Universal Robots PolyScope program: mt.urp

Program mt (installation=default directory=/programs createdIn=3.8.0.61336 lastSavedIn=3.8.0.61336 robotSerialNumber=2018359174)
Calibrated DH parameters: a=[0.000103, -0.165236, -0.391809, -0.000008, 0.000072, 0]; d=[0.08937, 126.180413, -125.613724, -0.456703, 0.094787, 0.082637]; alpha=[1.569508, -0.003108, -0.027037, 1.57048, -1.570735, 0]; deltaTheta=[0, -1.172139, 1.133037, 0.038915, 0.000034, 0.000049]
Robot Program (runOnlyOnce=false)
  var_1 := p[0.0,0.0,0.0,0.0,0.0,0.0]
  Plane_1 := p[0,0,0,0,0,0]
  Base := p[0,0,0,0,0,0]
  Script file /programs/X0.script
    | address="192.168.221.2"
    | port=3000
    | sname="mt"
    | socket_open(address,port,sname)
    | p=get_actual_tcp_pose()
    | socket_send_line("X0()",sname)
    | ret=socket_read_line(sname)
    | socket_close(sname)
    | if (ret != "OK"):
    |   popup(ret,title="X0",blocking=True)
    | end
  MoveJ speed 60 deg/s, acceleration 80 deg/s^2 (useActiveTCP=true)
    Waypoint CapturePoint_1: TCP in base x=190.539 y=-105.512 z=739.544 mm, rx=-2.169 ry=2.1248 rz=-0.097 rad; joints [0.073, -70.662, -54.312, -138.221, 90.524, 0.198] deg
  Wait Sleep waitTime=1
  Script file /programs/X1.script
    | address="192.168.221.2"
    | port=3000
    | sname="mt"
    | timeout=10
    | socket_open(address,port,sname)
    | p=get_actual_tcp_pose()
    | rpy=rotvec2rpy([p[3],p[4],p[5]])
    | socket_send_string("X1(",sname)
    | socket_send_string(p[0]*1000.,sname)
    | socket_send_string(",",sname)
    | socket_send_string(p[1]*1000.,sname)
    | socket_send_string(",",sname)
    | socket_send_string(p[2]*1000.,sname)
    | socket_send_string(",",sname)
    | socket_send_string(r2d(rpy[0]),sname)
    | socket_send_string(",",sname)
    | socket_send_string(r2d(rpy[1]),sname)
    | socket_send_string(",",sname)
    | socket_send_string(r2d(rpy[2]),sname)
    | socket_send_line(")",sname)
    | ret=socket_read_line(sname,timeout)
    | socket_close(sname)
    | if (ret != "OK"):
    |   popup(ret,title="X1",blocking=True)
    | end
  Wait Sleep waitTime=1
  Script file /programs/X2.script
    | address="192.168.221.2"
    | port=3000
    | sname="mt"
    | timeout=30
    | socket_open(address,port,sname)
    | socket_send_line("X2()",sname)
    | ret=socket_read_line(sname,timeout)
    | if (ret != "OK"):
    |   popup(ret,title="X2",blocking=True)
    | else:
    |   f=socket_read_ascii_float(6,sname,timeout)
    |   while (f[0]!=6):
    |     sleep(0.3)
    |     f=socket_read_ascii_float(6,sname,timeout)
    |   end
    |   rvec=rpy2rotvec([d2r(f[4]),d2r(f[5]),d2r(f[6])])
    |   counter=0
    |   while (counter<3):
    |     var_1[counter]=f[counter+1]/1000.
    |     counter=counter+1
    |   end
    |   counter=0
    |   while (counter<3):
    |     var_1[counter+3]=rvec[counter]
    |     counter=counter+1
    |   end
    | end
    | socket_close(sname)
  MoveL speed 250 mm/s, acceleration 1200 mm/s^2 (useActiveTCP=false) feature(featureName=Joint_0_name)
    Base := var_1
    Waypoint Waypoint_1: TCP in base x=190.558 y=-105.514 z=391.957 mm, rx=-2.1691 ry=2.1247 rz=-0.097 rad; joints [0.338, -45.209, -123.867, -94.129, 90.077, -0.554] deg
  Halt
